FUNCTION_BLOCK MulticastConveyorCTL (* Basic Function Block Type *)
  (* Standard: 61499-2 *)
  (* Version 0.2, 2003-12-04, JHC, Rockwell Automation, Renamed for better indexing. *)
  (* Version 0.1, 2002-11-05, JHC, Rockwell Automation, Corrected missing ST element in Algorithm REQ. *)
  (* Version 0.0, 2000-05-30, JHC, Rockwell Automation *)
  (* Compiler header: package fb.rt.cs725; *)
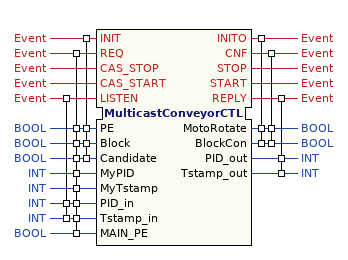
  EVENT_INPUT
    INIT WITH PE, Block, Candidate; (* Initialization Request *)
    REQ WITH PE, Block, Candidate, MyPID, MyTstamp, PID_in, Tstamp_in, MAIN_PE; (* Normal Execution Request *)
    CAS_STOP;
    CAS_START;
    LISTEN WITH PID_in, Tstamp_in;
  END_EVENT
  EVENT_OUTPUT
    INITO WITH MotoRotate, BlockCon; (* Initialization Confirm *)
    CNF WITH MotoRotate, BlockCon; (* Execution Confirmation *)
    STOP;
    START;
    REPLY WITH PID_out, Tstamp_out;
  END_EVENT
  VAR_INPUT
    PE : BOOL; (* Input event qualifier *)
    Block : BOOL;
    Candidate : BOOL;
    MyPID : INT;
    MyTstamp : INT;
    PID_in : INT;
    Tstamp_in : INT;
    MAIN_PE : BOOL;
  END_VAR
  VAR_OUTPUT
    MotoRotate : BOOL; (* Output event qualifier *)
    BlockCon : BOOL;
    PID_out : INT;
    Tstamp_out : INT;
  END_VAR
  VAR
    lastPE : BOOL := 1;
    lastBlock : BOOL := 0;
    MeFirst : BOOL;
    YouFirst : BOOL;
    LampClock : INT;
    DelayCounter : INT;
    DelayElapse : BOOL;
  END_VAR
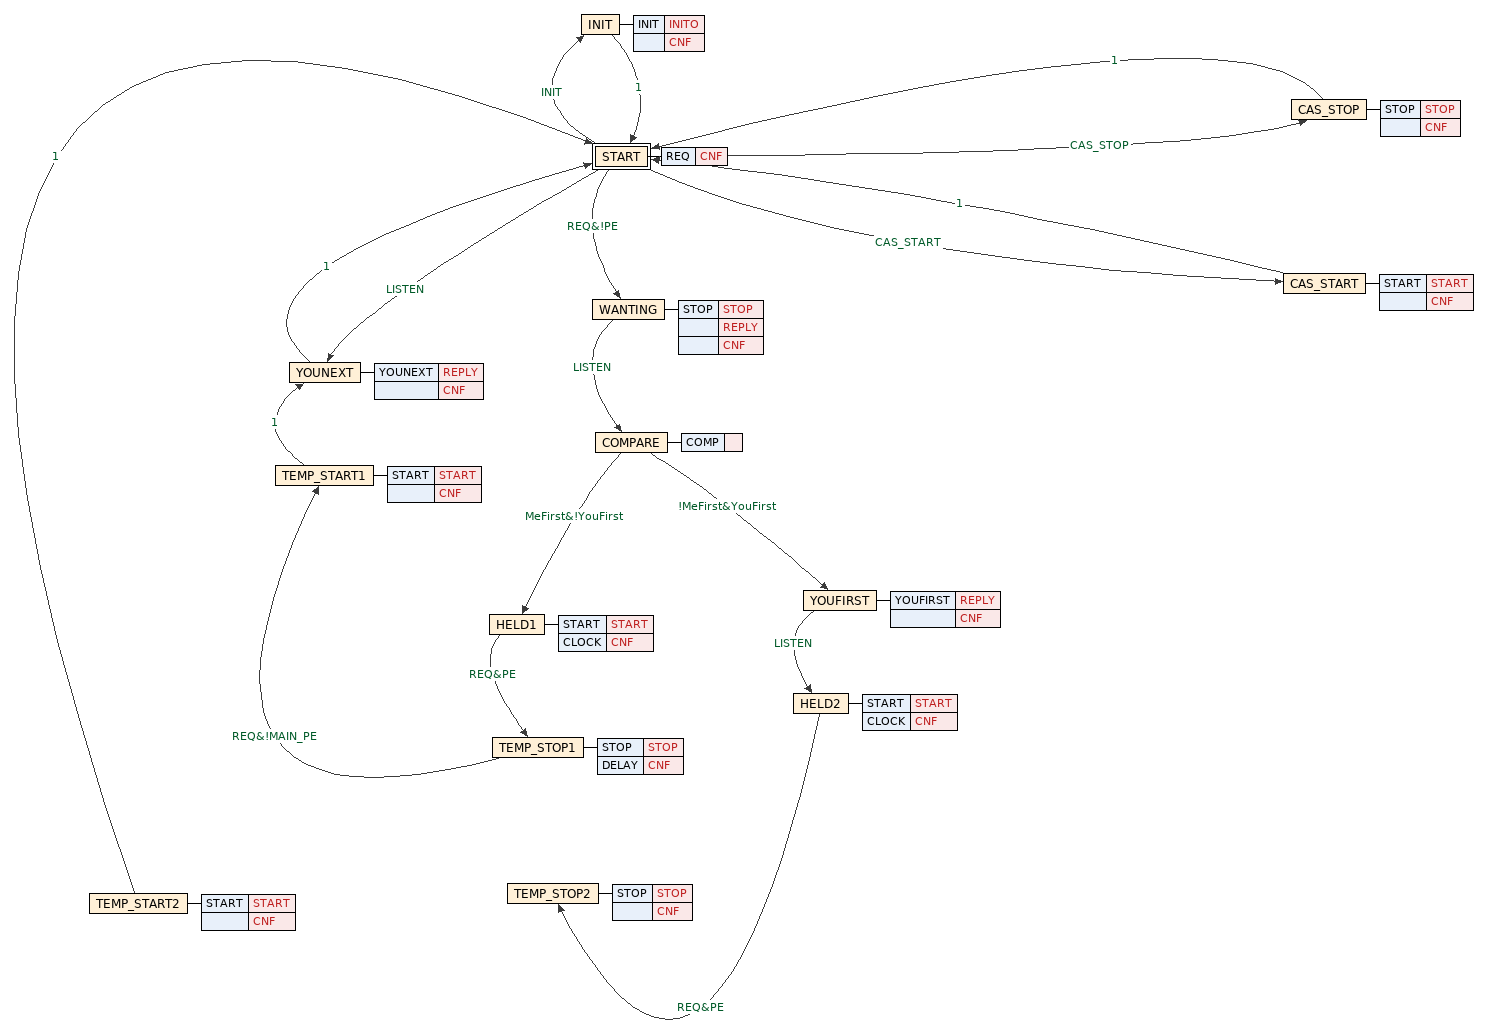
  EC_STATES
    START : REQ -> CNF; (* Initial State *)
    INIT : INIT -> INITO, -> CNF; (* Initialization *)
    CAS_START : START -> START, -> CNF;
    CAS_STOP : STOP -> STOP, -> CNF;
    WANTING : STOP -> STOP, -> REPLY, -> CNF;
    COMPARE : COMP;
    HELD1 : START -> START, CLOCK -> CNF;
    HELD2 : START -> START, CLOCK -> CNF;
    YOUFIRST : YOUFIRST -> REPLY, -> CNF;
    YOUNEXT : YOUNEXT -> REPLY, -> CNF;
    TEMP_STOP2 : STOP -> STOP, -> CNF;
    TEMP_START2 : START -> START, -> CNF;
    TEMP_STOP1 : STOP -> STOP, DELAY -> CNF;
    TEMP_START1 : START -> START, -> CNF;
  END_STATES
  EC_TRANSITIONS
    START TO INIT := INIT;
    INIT TO START := 1;
    START TO CAS_START := CAS_START;
    CAS_START TO START := 1;
    START TO CAS_STOP := CAS_STOP;
    CAS_STOP TO START := 1;
    START TO WANTING := REQ&!PE;
    WANTING TO COMPARE := LISTEN;
    YOUFIRST TO HELD2 := LISTEN;
    COMPARE TO YOUFIRST := !MeFirst&YouFirst;
    COMPARE TO HELD1 := MeFirst&!YouFirst;
    YOUNEXT TO START := 1;
    START TO YOUNEXT := LISTEN;
    HELD2 TO TEMP_STOP2 := REQ&PE;
    TEMP_START2 TO START := 1;
    HELD1 TO TEMP_STOP1 := REQ&PE;
    TEMP_STOP1 TO TEMP_START1 := REQ&!MAIN_PE;
    TEMP_START1 TO YOUNEXT := 1;
  END_TRANSITIONS
  ALGORITHM INIT IN Java: (* Initialization algorithm *)
System.out.println("In INT State");

MotoRotate.value=true;
Block.value=false;
LampClock.value=MyTstamp.value;
MeFirst.value=false;
YouFirst.value=false;

DelayElapse.value=false;
DelayCounter.value=0;

System.out.println(this+" "+MotoRotate.value);
System.out.println(MotoRotate.value);
  END_ALGORITHM
  ALGORITHM REQ IN Java: (* Normally executed algorithm *)
System.out.println("In REQ State");

MeFirst.value = false;
YouFirst.value = false;

DelayElapse.value=false;
DelayCounter.value=0;

LampClock.value++;
  END_ALGORITHM
  ALGORITHM START IN Java:
MotoRotate.value=true;
System.out.println(this+" Start "+MotoRotate.value);
  END_ALGORITHM
  ALGORITHM STOP IN Java:
MotoRotate.value=false;
System.out.println(this+" Stop "+MotoRotate.value);
  END_ALGORITHM
  ALGORITHM COMP IN Java:
System.out.println("In COMP State");
if(MyTstamp.value > Tstamp_in.value){
MeFirst.value = false;
YouFirst.value = true;
}else if (MyTstamp.value < Tstamp_in.value){
MeFirst.value = true;
YouFirst.value = false;
} else {
if(MyPID.value < PID_in.value){
MeFirst.value = false;
YouFirst.value = true;
} else {
MeFirst.value = true;
YouFirst.value = false;
}
}
  END_ALGORITHM
  ALGORITHM YOUFIRST IN Java:
System.out.println("In YOUFIRST State");
Tstamp_out.value = LampClock.value;
PID_out.value = MyPID.value;
  END_ALGORITHM
  ALGORITHM CLOCK IN Java:
System.out.println("Updating Clock");
LampClock.value = Tstamp_in.value;
  END_ALGORITHM
  ALGORITHM YOUNEXT IN Java:
System.out.println("In YOUNEXT State");
Tstamp_out.value = LampClock.value;
PID_out.value = MyPID.value;
  END_ALGORITHM
  ALGORITHM DELAY IN Java:
if(DelayCounter.value>10){
DelayElapse.value=true;
}else{
DelayCounter.value++;
}
  END_ALGORITHM
END_FUNCTION_BLOCK
